(* IEC 61131-3 sources: lacyccom/src/Blocks/Drives, 6 files *)

(* ---- Baseclass.st ---- *)
using System.Timer;
using Siemens.Simatic.DistributedIO;

NAMESPACE Simatic.Ax.LAcycCom

    CLASS ABSTRACT ReadWriteParameter
        VAR
            statrequestBuffer      : Resourcemanager;                                                                                                                  // Connection to the request buffer of the resource manager. All LAcycCom blocks have to use the same request buffer
            statdiagnostics        : LAcycCom_ooptypeDrivediagnostics;                                                                                                 // statdiagnostics structure
            statTimerStart         : BOOL := FALSE;                                                                                                                    // TRUE: Starts IEC-Timer
            statCmdBusy            : BOOL := FALSE;                                                                                                                    // TRUE: Process is NOT yet complete
            statCmdDone            : BOOL := FALSE;                                                                                                                    // TRUE: Data record was transferred
            statCmdError           : BOOL := FALSE;                                                                                                                    // TRUE: An error occurred during processing
            statHwId               : HW_IO := HW_IO#default;                                                                                                           // Intern hardware identifier of the hardware module
            statDoId               : INT;                                                                                                               // Intern identification number of the drive object
            statRefNo              : BYTE := BYTE#16#00;                                                                                                               // Reference number of request
            statFBState            : LAcycCom_ReadWriteStatus := LAcycCom_ReadWriteStatus#FB_IDLE;                                                                     // States in the function block state machine
            statFBSubState         : LAcycCom_ReadWriteStatus := LAcycCom_ReadWriteStatus#FB_BUSY_WRREC;                                                               // States in the function block during processing (busy state)
            statFBSubStateOld      : LAcycCom_ReadWriteStatus := LAcycCom_ReadWriteStatus#FB_BUSY_WRREC;                                                               // Previous state when temporary error occurs
            statStateNumber        : LAcycCom_ReadWriteStatus;                                                                                                         // State of the FB when error occurred
            statDatasetType        : SINT := SINT#0;                                                                                                                   // Dataset type used
            statStatus             : WORD := STATUS_NO_CALL;                                                                                                           // Static value for output status
            statSubfunctionStatus  : WORD := WORD#16#0000;                                                                                                             // Block status OR error information
            statErrorCount         : UINT := UINT#16#0000;                                                                                                             // Error counter of retry request
            statAllocatedIndex     : INT := -1;                                                                                                                        // Allocated element index in the buffer DB
            statCountOfElements    : INT := 0;                                                                                                                         // Number of parameters in the dataset
            statFirstParameterError: INT := -1;                                                                                                                        // Number of parameter at which the error occurred (-1: no parameter with error)
            statDataRecordNo       : DINT;                                                                                                                             // Used data record
            statReqParameter       : LAcycCom_TypestatstatReqParameter;                                                                                                // Request telegram
            statReqParameterInit   : LAcycCom_TypestatparameterAddress :=(attribute := BYTE#16#10, elementNo  := BYTE#16#01, parameterNo := UINT#0, index := UINT#0);

            statRespParameter: LAcycCom_TypestatRespParameter;  // Response telegram
            instWRREC        : WriteRecord;                     // WRREC command
            instRDREC        : ReadRecord;                      // RDREC command
            instIECTimer     : OnDelay;                         // IEC-Timer

            atmpSend : ARRAY[0..237]of BYTE ;
            atmpRec  : ARRAY[0..237]of BYTE ;

         END_VAR

         VAR CONSTANT
            DATA_TYPE_SILENT                    : SINT := SINT#1;        // LAcycCom_typeDriveSilentOperation is in use
            DATA_TYPE_DATASET_REAL              : SINT := SINT#2;        // LAcycCom_typeDriveDatasetReal is in use
            DATA_TYPE_DATASET_DWORD             : SINT := SINT#3;        // LAcycCom_typeDriveDatasetDWord is in use
            NO_PARAMETER_ERROR                  : INT  := INT#-1;        // No parameter error in response telegram
            ALL_ELEMENTS_OCCUPIED               : INT  := INT#-1;        // All buffer elements are occupied
            FORMAT_INTEGER_8                    : SINT := SINT#2;        // Identifier for Integer8 format
            FORMAT_INTEGER_16                   : SINT := SINT#3;        // Identifier for Integer16 format
            FORMAT_INTEGER_32                   : SINT := SINT#4;        // Identifier for Integer32 format
            FORMAT_UNSIGNED_8                   : SINT := SINT#5;        // Identifier for Unsigned8 format
            FORMAT_UNSIGNED_16                  : SINT := SINT#6;        // Identifier for Unsigned16 format
            FORMAT_UNSIGNED_32                  : SINT := SINT#7;        // Identifier for Unsigned32 format
            FORMAT_FLOATING_POINT               : SINT := SINT#8;        // Identifier for Floating Point format
            FORMAT_OCTET_STRING                 : SINT := SINT#10;       // Identifier for OctetString format
            FORMAT_TIME_DIFFERENCE              : SINT := SINT#13;       // Identifier for TimeDifference format
            FORMAT_ZERO                         : SINT := SINT#64;       // Identifier for void telegram
            FORMAT_BYTE                         : SINT := SINT#65;       // Identifier for BYTE format
            FORMAT_WORD                         : SINT := SINT#66;       // Identifier for WORD format
            FORMAT_DOUBLE_WORD                  : SINT := SINT#67;       // Identifier for Double WORD format
            FORMAT_ERROR                        : BYTE := BYTE#16#44;    // Identifier for a format error
            SILENT_OPERATION_PARA_UPPER_LIM     : INT  := 17;            // Maximum count of parameters when using Silent Operation PLC data type
            LENGTH_PARAMETER_TELEGRAM_UPPER_LIM : INT  := 233;           // Maximum length of telegram for parameter information in BYTE
            LENGTH_READ_TELEGRAM_UPPER_LIM      : INT  := 113;           // Maximum length of telegram for parameter information in BYTE
            MAX_ERROR_COUNT                     : UINT := UINT#40;       // Maximum error counter
            TIMER_TEMP_ERROR                    : LTime := T#200MS;       // Waiting time until next system function block call
            TIMER_ALLOCATION                    : LTime := T#10S;         // Timer limit for allocating a request element
            MAX_DRIVE_OBJECT_NO                 : INT  := 254;           // Maximum drive object number limited by SINAMICS p101
            STATUS_EXECUTION_FINISHED           : WORD := WORD#16#0000;  // Execution finished without errors
            STATUS_NO_CALL                      : WORD := WORD#16#7000;  // No call of FB
            STATUS_ALLOCATE                     : WORD := WORD#16#7001;  // FB is currently allocating a request element
            STATUS_GET_RESOURCE                 : WORD := WORD#16#7002;  // FB is waiting until it has “speaking rights”
            STATUS_BUSY                         : WORD := WORD#16#7003;  // FB is currently in processing
            STATUS_RELEASE                      : WORD := WORD#16#7004;  // FB is releasing the allocated element
            WARN_EXECUTE                        : WORD := WORD#16#7100;  // Execute input set during silent operation mode
            ERR_NO_OF_PARAMETERS                : WORD := WORD#16#8001;  // Invalid count of parameters
            ERR_INVALID_PRIORITY_CLASS          : WORD := WORD#16#8002;  // FB is NOT called in OB1
            ERR_REQUEST_REJECTED                : WORD := WORD#16#8004;  // Request rejected
            ERR_RESOURCE_RELEASED               : WORD := WORD#16#8005;  // Request is already released
            ERR_AMBIGUOUS_FB_CALL               : WORD := WORD#16#8006;  // Execute input set during processing (possible inconsistent data at output)
            ERR_INVALID_DATA_TYPE               : WORD := WORD#16#8200;  // Invalid PLC data type at the input "dataset"
            ERR_INVALID_BUF_INDEX               : WORD := WORD#16#8201;  // Buffer index is invalid
            ERR_INVALID_DRIVE_OBJECT_ID         : WORD := WORD#16#8208;  // Drive Object ID is out of range (Drive Object ID < 0 for local access, 1..254 for global access is allowed)
            ERR_COMMAND_TIMEOUT                 : WORD := WORD#16#8600;  // The assigned buffer element is no longer available for the request
            ERR_RDREC_TEMP_COUNTER              : WORD := WORD#16#8601;  // Counter for temporary errors reached the maximum during RDREC command
            ERR_WRREC_TEMP_COUNTER              : WORD := WORD#16#8602;  // Counter for temporary errors reached the maximum during WRREC command
            ERR_WRREC                           : WORD := WORD#16#8603;  // Error occurred during WRREC command
            ERR_RDREC                           : WORD := WORD#16#8604;  // Error occurred during RDREC command
            ERR_REFERENCE_NO                    : WORD := WORD#16#8605;  // Reference number of the request does NOT match the response reference number
            ERR_RESPONSE_ID                     : WORD := WORD#16#8606;  // Invalid response from the drive object
            ERR_PARAMETER_NO                    : WORD := WORD#16#8607;  // The number of parameters received does NOT match the requested number of parameters
            ERR_DRIVE_OBJECT_NO                 : WORD := WORD#16#8608;  // The drive object does NOT match the responded drive object
            ERR_ALLOCATION_TIME                 : WORD := WORD#16#8609;  // The allocation time exceeded the configured value
            ERR_MOVE_BLK_VARIANT                : WORD := WORD#16#8610;  // Error occurred during MOVE_BLK_VARIANT command
            ERR_UNDEFINED_STATE                 : WORD := WORD#16#8611;  // Error due to an undefined state
            ERR_UNDEFINED_SUBSTATE              : WORD := WORD#16#8612;  // Error due to an undefined substate
            ERR_PARAMETER                       : WORD := WORD#16#8619;  // Error in at least one parameter (see: errorValue in dataset)
         END_VAR

        METHOD ABSTRACT BUSY END_METHOD

        METHOD PUBLIC FINAL execute

            //----------------------------------------------------------------------
            // State Machine
            //----------------------------------------------------------------------

            IF NOT (statFBState = LAcycCom_ReadWriteStatus#FB_IDLE OR
                    statFBState = LAcycCom_ReadWriteStatus#FB_DONE OR
                    statFBState = LAcycCom_ReadWriteStatus#FB_ERROR ) THEN  // Functionality running
              CASE statFBState OF
                LAcycCom_ReadWriteStatus#FB_FIRST_CYCLE:  // First cycle state

                    THIS.FIRST_CYCLE();

                    LAcycCom_ReadWriteStatus#FB_ALLOCATE:

                    THIS.Allocate();

                LAcycCom_ReadWriteStatus#FB_GET_RESOURCE:

                    THIS.GET_RESOURCE();

                LAcycCom_ReadWriteStatus#FB_BUSY:

                    THIS.BUSY();

                LAcycCom_ReadWriteStatus#FB_RELEASE:

                    THIS.RELEASE();

                ELSE
                  statStatus := ERR_UNDEFINED_STATE;
                  statStateNumber := statFBState;
                  statFBState := LAcycCom_ReadWriteStatus#FB_ERROR;
              END_CASE;

            END_IF;

            //----------------------------------------------------------------------
            // Error handling and write outputs
            //----------------------------------------------------------------------

            IF (statFBState = LAcycCom_ReadWriteStatus#FB_ERROR) THEN
              // Release the allocated element when error occurs
              IF (statStateNumber <> LAcycCom_ReadWriteStatus#FB_FIRST_CYCLE) AND (statStateNumber <> LAcycCom_ReadWriteStatus#FB_ALLOCATE)
              THEN
                statrequestBuffer.release(statAllocatedIndex);
              END_IF;
              statdiagnostics.stateNumber := statStateNumber;
              statdiagnostics.subfunctionStatus := statSubfunctionStatus;
              statdiagnostics.status := statStatus;

            END_IF;

        END_METHOD

        METHOD FINAL FIRST_CYCLE
            VAR_TEMP
                tempLoopIndex : INT;
                tempVoidDiagnostics : LAcycCom_ooptypeDriveDiagnostics;   // Temporary empty diagnostics structure
                tempVoidHeader : LAcycCom_Typestatheader;   // Temporary empty header structure
             END_VAR

              // Clearing the sending buffer
              statReqParameter.header := tempVoidHeader;
              FOR tempLoopIndex := 0 TO LAcycComConstantsInt#LACYCCOM_READ_PARAMETERS_UPPER_LIM DO
                statReqParameter.parameterAddress[tempLoopIndex] := statReqParameterInit;
              END_FOR;

              // Clearing the receive buffer
              statRespParameter.header := tempVoidHeader;
              FOR tempLoopIndex := 0 TO LENGTH_PARAMETER_TELEGRAM_UPPER_LIM DO
                statRespParameter.data[tempLoopIndex] := BYTE#16#00;
              END_FOR;

              // Initialization after start, depending on the used PLC data type

                IF statDoId < 0 THEN // V1.5
                  statDataRecordNo := 16#B02E; // Base Mode Parameter Access local; doId NOT relevant
                  statDoId := 0; //set DO to zero for use in header
                ELSIF (statDoId <= MAX_DRIVE_OBJECT_NO)
                  AND (statDoId <> 0)
                THEN // V1.5.2
                  statDataRecordNo := 47; // Data record 47; Base Mode Parameter Access global

                ELSE // V1.5.2
                  // Wrong drive object ID at input
                  statStateNumber := statFBState;
                  statStatus := ERR_INVALID_DRIVE_OBJECT_ID;
                  statFBState := LAcycCom_ReadWriteStatus#FB_ERROR;
                END_IF;

                statHwId := statHwId;

              statdiagnostics := tempVoidDiagnostics;
              IF statStatus = WARN_EXECUTE THEN
                statdiagnostics.status := statStatus;
              END_IF;

              statdiagnostics.driveObjectId       := TO_USINT(statDoId);
              statdiagnostics.hardwareId          := statHwId;
              statdiagnostics.firstParameterError := statFirstParameterError;  // V1.3.2
              statdiagnostics.errorValue          := BYTE#16#FF;               // V1.3.2

              // Reference number for next request
              statRefNo := to_byte(to_int(statRefNo) + INT#1);

              IF statFBState = LAcycCom_ReadWriteStatus#FB_ERROR THEN // V1.5.2: Check IF error appeared
                ;

              // Next state is depending on the FB mode
            ELSE
                statStatus := STATUS_ALLOCATE;
                statFBState := LAcycCom_ReadWriteStatus#FB_ALLOCATE;

            END_IF;

        END_METHOD

        METHOD FINAL Allocate
                  // Allocation of a request element
                  statAllocatedIndex := statrequestBuffer.allocate(hardwareId :=statHwId);

                  IF statAllocatedIndex >= 0 THEN

                    statTimerStart := FALSE;
                    statStatus := STATUS_GET_RESOURCE;
                    statFBState := LAcycCom_ReadWriteStatus#FB_GET_RESOURCE;

                  ELSIF (instIECTimer.output = TRUE) THEN
                    statStateNumber := statFBState;
                    statStatus := ERR_ALLOCATION_TIME;
                    statFBState := LAcycCom_ReadWriteStatus#FB_ERROR;

                  ELSE
                    ; // Waiting until lockbit is reset and a request element is available
                  END_IF; // (buffer.lockBuffer = FALSE) AND (buffer.actualWriteIndex >= 0)

                  instIECTimer(signal := statTimerStart,
                                duration := TIMER_ALLOCATION);

                  statTimerStart := TRUE;
                  IF (instIECTimer.output = TRUE) THEN
                    statTimerStart := FALSE;
                  END_IF;
        END_METHOD

        METHOD FINAL GET_RESOURCE
            CASE statrequestBuffer.GetRessource(statAllocatedIndex) of
                // Check buffer index for correctness
                LAcycCom_ResourceManagerRetval#ERR_INVALID_BUF_INDEX:
                  statStateNumber := statFBState;
                  statStatus := ERR_INVALID_BUF_INDEX;
                  statFBState := LAcycCom_ReadWriteStatus#FB_ERROR;

                LAcycCom_ResourceManagerRetval#ERR_REQUEST_REJECTED:
                    // Request was rejected by buffer manager
                    statStateNumber := statFBState;
                    statStatus := ERR_REQUEST_REJECTED;
                    statFBState := LAcycCom_ReadWriteStatus#FB_ERROR;

                LAcycCom_ResourceManagerRetval#ERR_RESOURCE_RELEASED:
                    // Request already released
                    statStateNumber := statFBState;
                    statStatus := ERR_RESOURCE_RELEASED;
                    statFBState := LAcycCom_ReadWriteStatus#FB_ERROR;

                LAcycCom_ResourceManagerRetval#STATUS_BUSY:
                    // Element is enabled
                    statStatus := STATUS_BUSY;
                    statFBState := LAcycCom_ReadWriteStatus#FB_BUSY;
                    statFBSubState := LAcycCom_ReadWriteStatus#FB_GET_SUBSTATE;

                LAcycCom_ResourceManagerRetval#STATUS_GET_RESOURCE:
                    // Element NOT enabled yet
                    //
                    statStatus := STATUS_GET_RESOURCE;
                ELSE
                  ;
                END_CASE;
        end_Method

        METHOD FINAL RELEASE
                  CASE statrequestBuffer.release(statAllocatedIndex) of
                    LAcycCom_ResourceManagerRetval#ERR_INVALID_BUF_INDEX:
                      statStatus := ERR_INVALID_BUF_INDEX;
                      statStateNumber := statFBState;
                      statFBState := LAcycCom_ReadWriteStatus#FB_ERROR;

                    LAcycCom_ResourceManagerRetval#STATUS_EXECUTION_FINISHED:
                      statStatus := STATUS_EXECUTION_FINISHED;
                      statFBState := LAcycCom_ReadWriteStatus#FB_DONE;
                  ELSE
                    ;
                  END_CASE;
        end_Method

        Method PUBLIC FINAL errorDiagnostics   : LAcycCom_ooptypeDrivediagnostics;
            errorDiagnostics := statdiagnostics;
        End_Method

        Method PUBLIC FINAL Status   : LAcycComstateDef;
            CASE statFBState OF
                LAcycCom_ReadWriteStatus#FB_IDLE:
                    Status := LAcycComstateDef#IDLE;

                LAcycCom_ReadWriteStatus#FB_FIRST_CYCLE,
                LAcycCom_ReadWriteStatus#FB_ALLOCATE,
                LAcycCom_ReadWriteStatus#FB_GET_RESOURCE,
                LAcycCom_ReadWriteStatus#FB_BUSY,
                LAcycCom_ReadWriteStatus#FB_RELEASE:
                    Status := LAcycComstateDef#BUSY;

                LAcycCom_ReadWriteStatus#FB_DONE:
                    Status := LAcycComstateDef#DONE;

                LAcycCom_ReadWriteStatus#FB_ERROR:
                    Status := LAcycComstateDef#Error;

                ELSE
                ;
            END_CASE;
        End_Method

        METHOD PUBLIC FINAL Config : BOOL
          VAR_INPUT
              requestBuffer : Resourcemanager;   // Connection to the request buffer of the resource manager. All LAcycCom blocks have to use the same request buffer
           END_VAR

           IF requestBuffer <> NULL THEN
            statrequestBuffer := requestBuffer;
            Config := TRUE;
           ELSE
            ;
           END_IF;

      END_METHOD
    END_CLASS

END_NAMESPACE

(* ---- classReadDriveParams.st ---- *)
using System.Timer;
using siemens.Simatic.DistributedIO;

NAMESPACE Simatic.Ax.LAcycCom
    CLASS LAcycCom_classReadDriveParams EXTENDS ReadWriteParameter
        VAR PRIVATE
            statparameterCount: INT := -1;
            dataset           : Array[0..LAcycComConstantsInt#LACYCCOM_READ_PARAMETERS_UPPER_LIM] of LAcycCom_typeDriveDataset;          // Dataset with all parameters to be read
            statParameter     : Array[0..LAcycComConstantsInt#LACYCCOM_READ_PARAMETERS_UPPER_LIM] of LAcycCom_TypestatstatParameter;     // Parameter dataset
            parameterAddress  : Array[0..LAcycComConstantsInt#LACYCCOM_READ_PARAMETERS_UPPER_LIM] of LAcycCom_TypestatparameterAddress;  // Parameter data in telegram
          END_VAR

        METHOD OVERRIDE BUSY
            VAR_TEMP
                tempCmdValid         : BOOL;                       // TRUE: New data record was received and is valid
                tempStatusWord       : WORD;                       // Temporary status
                tempWord             : WORD;                       // Temporary WORD variable
                tempPointer          : INT;                        // Temporary pointer variable
                tempLoopIndex        : INT;                        // Temporary loop index variable
                tempBlkVariant       : INT;                        // Temporary result of MOVE_BLK_VARIANT
                tempCmdStatus        : DWORD;                      // Temporary status of WRREC and RDREC command
                tempDWord            : DWORD;                      // Temporary DWORD variable
                tempActualElementReal: LAcycCom_typeDriveDataset;  // Temporary element of the dataset (REAL values)
             END_VAR

            IF (statrequestBuffer.GetRessource(statAllocatedIndex)=LAcycCom_ResourceManagerRetval#STATUS_BUSY)
                THEN
                  CASE statFBSubState OF
                    LAcycCom_ReadWriteStatus#FB_GET_SUBSTATE:
                      statFBSubState := LAcycCom_ReadWriteStatus#FB_BUSY_WRREC;

                    LAcycCom_ReadWriteStatus#FB_BUSY_WRREC:  // Writing the dataset configuration into the drive object

                      IF (statCmdBusy = FALSE) THEN
                        // Resets WRREC command
                        instWRREC(request := FALSE,
                                  RECORD := THIS.atmpRec);
                        // Creating header data
                        statReqParameter.header.refNo := statRefNo; // Telegram reference number
                        statReqParameter.header.reqId := BYTE#16#01;  // 0x01 = request parameters
                        statReqParameter.header.doId := TO_BYTE(statDoId);  // Drive object identification number
                        statReqParameter.header.parameterNo := TO_BYTE(statCountOfElements);  // Count of parameters

                        // Copying the dataset into a static variable (depending on the used PLC data type)

                          FOR tempLoopIndex := 0 TO statCountOfElements - 1 DO
                            tempActualElementReal := dataset[tempLoopIndex];

                            statParameter[tempLoopIndex].index := tempActualElementReal.index;
                            statParameter[tempLoopIndex].parameterNo := tempActualElementReal.parameterNumber;
                            statReqParameter.parameterAddress[tempLoopIndex].parameterNo := statParameter[tempLoopIndex].parameterNo;  // Parameter number
                            statReqParameter.parameterAddress[tempLoopIndex].index := statParameter[tempLoopIndex].index;  // Subindex of parameter
                         END_FOR;

                      END_IF; // statCmdBusy = FALSE
                      SerializeBig(UINT#0,
                                  statReqParameter,
                                  THIS.atmpSend );
                      // WRREC command
                      instWRREC(REQUEST := TRUE,                                                 // Transfer data record
                                 hardwareID := statHwId,           // ID number of the hardware component
                                 INDEX  := statDataRecordNo,   // Data record number
                                 LENGTH := UINT#0,             // Maximum length of the data record to be transferred in bytes
                                 DONE   => statCmdDone,        // Data record was transferred
                                 BUSY   => statCmdBusy,        // The writing process is NOT yet complete
                                 ERROR  => statCmdError,       // An error occurred during the writing process
                                 STATUS => tempCmdStatus,      // Status[1] = Error => Status[2] Error Decode + Status[3] Error Code
                                 RECORD := THIS.atmpSend);     // Data record

                      // Error occurred
                      IF (statCmdError = TRUE) AND NOT(statFBState = LAcycCom_ReadWriteStatus#FB_ERROR) THEN
                        tempStatusWord.%B0 := tempCmdStatus.%B1;
                        tempStatusWord.%B1 := tempCmdStatus.%B2;

                        //Temporary command status (80A1, 80A7, 80B5, 80C0, 80C1, 80C2, 80C3 oder 80C4) are valid and retry command
                        IF (tempStatusWord = WORD#16#80A1) OR  // Negative acknowledgment when writing to the module
                          (tempStatusWord = WORD#16#80A7) OR   // DP slave OR module is occupied (temporary error)
                          (tempStatusWord = WORD#16#80B5) OR   // DP slave OR module NOT ready
                          (tempStatusWord = WORD#16#80C0) OR   // The data can only be written when the CPU is in STOP mode. Note: this means that writing by the user program is NOT possible. You can only write the data online with PG/PC.
                          (tempStatusWord = WORD#16#80C1) OR   // The data of the previous write job on the module for the same data record have NOT yet been processed by the module.
                          (tempStatusWord = WORD#16#80C2) OR   // The module is currently processing the maximum possible number of jobs for a CPU.
                          (tempStatusWord = WORD#16#80C3) OR   // The required operating resources are currently occupied.
                          (tempStatusWord = WORD#16#80C4) THEN // Internal temporary error. Job could NOT be executed. Repeat the job. IF this error occurs often, check your installation for sources of electrical interference.

                          IF (statErrorCount >= MAX_ERROR_COUNT) THEN
                            statStateNumber := statFBSubState;
                            statSubfunctionStatus := tempStatusWord;
                            statStatus := ERR_WRREC_TEMP_COUNTER;
                            statFBState := LAcycCom_ReadWriteStatus#FB_ERROR;
                          ELSE
                            statErrorCount := statErrorCount + UINT#1;  // Increment internal error counter
                            statFBSubStateOld := LAcycCom_ReadWriteStatus#FB_BUSY_WRREC;
                            statFBSubState := LAcycCom_ReadWriteStatus#FB_BUSY_WAIT;
                          END_IF;
                        ELSE
                          statStateNumber := statFBSubState;
                          statSubfunctionStatus := tempStatusWord;
                          statStatus := ERR_WRREC;
                          statFBState := LAcycCom_ReadWriteStatus#FB_ERROR;
                        END_IF;

                      ELSIF (statCmdDone = TRUE) AND NOT(statFBState = LAcycCom_ReadWriteStatus#FB_ERROR) THEN  // Processing completed without errors
                        statErrorCount := UINT#0;  // V1.5.1 Reset error counter
                        statFBSubState := LAcycCom_ReadWriteStatus#FB_BUSY_RDREC; // WRREC completed and continue with RDREC
                      END_IF; // statCmdError = TRUE

                      LAcycCom_ReadWriteStatus#FB_BUSY_RDREC:  // Reading the values from the drive object
                      // Resets RDREC command
                      IF (statCmdBusy = FALSE) THEN
                        instRDREC(REQUEST := FALSE,
                                   RECORD := THIS.atmpRec);
                      END_IF;

                      instRDREC(REQUEST := TRUE,                                                 // Transfer data record
                                 hardwareID := statHwId,           // ID number of the hardware component
                                 INDEX      := statDataRecordNo,   // Data record number
                                 MAXLENGTH  := UINT#0,             // Maximum length in bytes of the data record information to be read
                                 VALID      => tempCmdValid,       // New data record was received and is valid
                                 BUSY       => statCmdBusy,        // The reading process is NOT yet complete
                                 ERROR      => statCmdError,       // An error occurred during the reading process
                                 STATUS     => tempCmdStatus,      // Status[1] = Error => Status[2] Error Decode + Status[3] Error Code
                                 RECORD     := THIS.atmpRec);      // Destination area for the data record read

                      DeserializeBig(UINT#0,
                                 THIS.atmpRec,
                                 statRespParameter);
                      // Error occurred
                      IF (statCmdError = TRUE) THEN
                        // Get the error information from the status information
                        tempStatusWord.%B0 := tempCmdStatus.%B1;
                        tempStatusWord.%B1 := tempCmdStatus.%B2;

                        //Temporary command status (80A0, 80A7, 80B5, 80C0, 80C1, 80C2, 80C3 oder 80C4) are valid and retry command
                        IF (tempStatusWord = WORD#16#80A0) OR  // Negative acknowledgment when reading the module
                          (tempStatusWord = WORD#16#80A7) OR   // DP slave OR module is occupied (temporary error)
                          (tempStatusWord = WORD#16#80B5) OR   // DP slave OR module NOT ready
                          (tempStatusWord = WORD#16#80C0) OR   // The data can only be written when the CPU is in STOP mode. Note: this means that writing by the user program is NOT possible. You can only write the data online with PG/PC.
                          (tempStatusWord = WORD#16#80C1) OR   // The data of the previous write job on the module for the same data record have NOT yet been processed by the module.
                          (tempStatusWord = WORD#16#80C2) OR   // The module is currently processing the maximum possible number of jobs for a CPU.
                          (tempStatusWord = WORD#16#80C3) OR   // The required operating resources are currently occupied.
                          (tempStatusWord = WORD#16#80C4) THEN // Internal temporary error. Job could NOT be executed. Repeat the job. IF this error occurs often, check your installation for sources of electrical interference.

                          IF (statErrorCount >= MAX_ERROR_COUNT) THEN
                            statStateNumber := statFBSubState;
                            statSubfunctionStatus := tempStatusWord;
                            statStatus := ERR_RDREC_TEMP_COUNTER;
                            statFBState := LAcycCom_ReadWriteStatus#FB_ERROR;
                          ELSE
                            statErrorCount := statErrorCount + UINT#1;  // Increment internal error counter
                            statFBSubStateOld := LAcycCom_ReadWriteStatus#FB_BUSY_RDREC;
                            // V1.3.2. IF error 80A0 THEN should be retry with WRREC command
                            IF (tempStatusWord = WORD#16#80A0) THEN
                              statFBSubStateOld := LAcycCom_ReadWriteStatus#FB_BUSY_WRREC;
                            END_IF;
                            statFBSubState := LAcycCom_ReadWriteStatus#FB_BUSY_WAIT;
                          END_IF; // statErrorCount >= MAX_ERROR_COUNT
                        ELSE
                          statStateNumber := statFBSubState;
                          statSubfunctionStatus := tempStatusWord;
                          statStatus := ERR_RDREC;
                          statFBState := LAcycCom_ReadWriteStatus#FB_ERROR;
                        END_IF;

                        // Error : Reference number of the request does NOT match with the response reference number
                      ELSIF (statCmdBusy = FALSE) AND
                        (statRefNo <> statRespParameter.header.refNo) AND
                        (tempCmdValid = TRUE) THEN

                        statStateNumber := statFBSubState;
                        statStatus := ERR_REFERENCE_NO;
                        statFBState := LAcycCom_ReadWriteStatus#FB_ERROR;

                        // Error : Invalid response from the drive object (reqId: 16#01 - reading parameter successful; 16#81: reading parameter finished with error)
                      ELSIF NOT (statRespParameter.header.reqId = BYTE#16#81 OR statRespParameter.header.reqId = BYTE#16#01) AND
                        (statCmdBusy = FALSE) AND
                        (tempCmdValid = TRUE) THEN
                        statStateNumber := statFBSubState;
                        statStatus := ERR_RESPONSE_ID;
                        statFBState := LAcycCom_ReadWriteStatus#FB_ERROR;

                        // Error : The received number of parameters does NOT match with the requested number of parameters
                      ELSIF (statCmdBusy = FALSE) AND
                        (statCountOfElements <> TO_INT(statRespParameter.header.parameterNo)) AND
                        (tempCmdValid = TRUE) THEN

                        statStateNumber := statFBSubState;
                        statStatus := ERR_PARAMETER_NO;
                        statFBState := LAcycCom_ReadWriteStatus#FB_ERROR;

                        // Error : The drive object does NOT match with the responsed DO
                      ELSIF (statCmdBusy = FALSE) AND
                        (TO_BYTE(statDoId) <> statRespParameter.header.doId) AND
                        (tempCmdValid = TRUE) THEN

                        statStateNumber := statFBSubState;
                        statStatus := ERR_DRIVE_OBJECT_NO;
                        statFBState := LAcycCom_ReadWriteStatus#FB_ERROR;

                        // No error occurred during reading parameters
                      ELSIF (tempCmdValid = TRUE) THEN
                        // Analyse of the response buffer
                        tempPointer := 0;
                        FOR tempLoopIndex := 0 TO statCountOfElements - 1 DO
                          statParameter[tempLoopIndex].format := statRespParameter.data[tempPointer];  // Format of the parameter

                          // Format = Error
                          IF (((TO_SINT(statRespParameter.data[tempPointer]) > FORMAT_DOUBLE_WORD) OR
                            ((TO_SINT(statRespParameter.data[tempPointer]) > FORMAT_FLOATING_POINT) AND (TO_SINT(statRespParameter.data[tempPointer]) < FORMAT_OCTET_STRING)) OR
                            ((TO_SINT(statRespParameter.data[tempPointer]) > FORMAT_OCTET_STRING) AND (TO_SINT(statRespParameter.data[tempPointer]) < FORMAT_TIME_DIFFERENCE)) OR
                            ((TO_SINT(statRespParameter.data[tempPointer]) > FORMAT_TIME_DIFFERENCE) AND (TO_SINT(statRespParameter.data[tempPointer]) < FORMAT_BYTE)) OR
                            (TO_SINT(statRespParameter.data[tempPointer]) < FORMAT_INTEGER_8))) AND (TO_SINT(statRespParameter.data[tempPointer]) <> FORMAT_ZERO)
                          THEN

                            // Format = Error, summarize the first and second error BYTE in a WORD error variable for each parameter
                            statParameter[tempLoopIndex].errorValue := statRespParameter.data[tempPointer + 3];
                            IF (statFirstParameterError = NO_PARAMETER_ERROR) THEN
                              statdiagnostics.firstParameterError := tempLoopIndex;
                              statdiagnostics.errorValue := statParameter[tempLoopIndex].errorValue; // V1.3.2
                              statFirstParameterError := tempLoopIndex;
                              statStateNumber := statFBSubState;
                              statStatus := ERR_PARAMETER;
                              statFBState := LAcycCom_ReadWriteStatus#FB_ERROR;
                            END_IF;
                            // Points to the next parameter address
                            tempPointer := tempPointer + 6;

                          ELSE

                            CASE TO_SINT(statRespParameter.data[tempPointer]) OF
                              FORMAT_INTEGER_8:

                                  statParameter[tempLoopIndex].realValue := TO_REAL(TO_SINT(statRespParameter.data[tempPointer + 2]));
                                  statParameter[tempLoopIndex].dwordValue := statRespParameter.data[tempPointer + 2];

                                statParameter[tempLoopIndex].errorValue := BYTE#16#FF; // Sets the error status and diagnostics
                                tempPointer := tempPointer + 4; // Points to the next parameter address

                              FORMAT_INTEGER_16:
                                tempWord.%B0 := statRespParameter.data[tempPointer + 3];
                                tempWord.%B1 := statRespParameter.data[tempPointer + 2];

                                statParameter[tempLoopIndex].realValue := TO_REAL(TO_INT(tempWord));
                                statParameter[tempLoopIndex].dwordValue := tempWord;
                                statParameter[tempLoopIndex].errorValue := BYTE#16#FF; // Sets the error status and diagnostics
                                tempPointer := tempPointer + 4; // Points to the next parameter address

                              FORMAT_INTEGER_32:
                                tempDWord.%B0 := statRespParameter.data[tempPointer + 5];
                                tempDWord.%B1 := statRespParameter.data[tempPointer + 4];
                                tempDWord.%B2 := statRespParameter.data[tempPointer + 3];
                                tempDWord.%B3 := statRespParameter.data[tempPointer + 2];

                                statParameter[tempLoopIndex].realValue := TO_REAL(TO_DINT(tempDWord));
                                statParameter[tempLoopIndex].dwordValue := tempDWord;

                                statParameter[tempLoopIndex].errorValue := BYTE#16#FF; // Sets the error status and diagnostics
                                tempPointer := tempPointer + 6; // Points to the next parameter address

                              FORMAT_UNSIGNED_8, FORMAT_OCTET_STRING: // V1.5 change OCTET_STRING

                                statParameter[tempLoopIndex].realValue := TO_REAL(TO_USINT(statRespParameter.data[tempPointer + 2]));
                                statParameter[tempLoopIndex].dwordValue := statRespParameter.data[tempPointer + 2];

                                statParameter[tempLoopIndex].errorValue := BYTE#16#FF; // Sets the error status and diagnostics
                                tempPointer := tempPointer + 4; // Points to the next parameter address
                              FORMAT_UNSIGNED_16:
                                tempWord.%B0 := statRespParameter.data[tempPointer + 3];
                                tempWord.%B1 := statRespParameter.data[tempPointer + 2];

                                statParameter[tempLoopIndex].realValue := TO_REAL(TO_UINT(tempWord));
                                statParameter[tempLoopIndex].dwordValue := tempWord;

                                statParameter[tempLoopIndex].errorValue := BYTE#16#FF; // Sets the error status and diagnostics
                                tempPointer := tempPointer + 4; // Points to the next parameter address

                              FORMAT_UNSIGNED_32, FORMAT_TIME_DIFFERENCE:
                                tempDWord.%B0 := statRespParameter.data[tempPointer + 5];
                                tempDWord.%B1 := statRespParameter.data[tempPointer + 4];
                                tempDWord.%B2 := statRespParameter.data[tempPointer + 3];
                                tempDWord.%B3 := statRespParameter.data[tempPointer + 2];

                                statParameter[tempLoopIndex].realValue := TO_REAL(TO_UDINT(tempDWord));
                                statParameter[tempLoopIndex].dwordValue := tempDWord;

                                statParameter[tempLoopIndex].errorValue := BYTE#16#FF; // Sets the error status and diagnostics
                                tempPointer := tempPointer + 6; // Points to the next parameter address

                              FORMAT_FLOATING_POINT, FORMAT_DOUBLE_WORD:
                                tempDWord.%B0 := statRespParameter.data[tempPointer + 5];
                                tempDWord.%B1 := statRespParameter.data[tempPointer + 4];
                                tempDWord.%B2 := statRespParameter.data[tempPointer + 3];
                                tempDWord.%B3 := statRespParameter.data[tempPointer + 2];

                                statParameter[tempLoopIndex].realValue := TO_REAL(tempDWord);
                                statParameter[tempLoopIndex].dwordValue := tempDWord;

                                statParameter[tempLoopIndex].errorValue := BYTE#16#FF; // Sets the error status and diagnostics
                                tempPointer := tempPointer + 6; // Points to the next parameter address

                              FORMAT_BYTE:
                                statParameter[tempLoopIndex].realValue := TO_REAL(TO_DWORD(statRespParameter.data[tempPointer + 2]));
                                statParameter[tempLoopIndex].dwordValue := statRespParameter.data[tempPointer + 2];

                                statParameter[tempLoopIndex].errorValue := BYTE#16#FF; // Sets the error status and diagnostics
                                tempPointer := tempPointer + 4; // Points to the next parameter address

                              FORMAT_WORD:
                                tempWord.%B0 := statRespParameter.data[tempPointer + 3];
                                tempWord.%B1 := statRespParameter.data[tempPointer + 2];

                                statParameter[tempLoopIndex].realValue := TO_REAL(TO_DWORD(tempWord));
                                statParameter[tempLoopIndex].dwordValue := tempWord;

                                statParameter[tempLoopIndex].errorValue := BYTE#16#FF; // Sets the error status and diagnostics
                                tempPointer := tempPointer + 4; // Points to the next parameter address

                              ELSE
                                ;
                            END_CASE;

                          END_IF; // Format = Error
                        END_FOR; // Analyse of the response buffer

                        // Copying parameter data into the dataset (depending on the used PLC data type)

                          FOR tempLoopIndex := 0 TO statCountOfElements - 1 BY 1 DO
                            tempActualElementReal.index := statParameter[tempLoopIndex].index;
                            tempActualElementReal.parameterNumber := statParameter[tempLoopIndex].parameterNo;
                            tempActualElementReal.Rvalue := statParameter[tempLoopIndex].realValue;
                            tempActualElementReal.DWvalue := statParameter[tempLoopIndex].dwordValue;
                            tempActualElementReal.errorValue := statParameter[tempLoopIndex].errorValue;
                           // tempBlkVariant := MOVE_BLK_VARIANT(SRC := tempActualElementReal, COUNT := 1, SRC_INDEX := 0, DEST_INDEX := tempLoopIndex, DEST => dataset);
                            dataset[tempLoopIndex] := tempActualElementReal;
                            // Error occurred during MOVE_BLK_VARIANT command
                            IF (tempBlkVariant <> 0) THEN
                              statStateNumber := statFBSubState;
                              statSubfunctionStatus := TO_WORD(tempBlkVariant);
                              statStatus := ERR_MOVE_BLK_VARIANT;
                              statFBState := LAcycCom_ReadWriteStatus#FB_ERROR;
                              statdiagnostics.firstParameterError := tempLoopIndex;
                            END_IF;
                          END_FOR;

                        // Next state is depending on the FB mode
                        IF NOT(statFBState = LAcycCom_ReadWriteStatus#FB_ERROR) THEN
                          statStatus := STATUS_RELEASE;
                          statFBState := LAcycCom_ReadWriteStatus#FB_RELEASE;

                        END_IF; // statMode = MODE_WITH_BUFFER_MANAGER
                      END_IF; // statCmdError = TRUE

                      LAcycCom_ReadWriteStatus#FB_BUSY_WAIT:
                      // Timer for temporary errors
                      instIECTimer(signal := statTimerStart,
                                    duration := TIMER_TEMP_ERROR);

                      statTimerStart := TRUE;
                      IF (instIECTimer.output = TRUE) THEN
                        statTimerStart := FALSE;
                        statFBSubState := statFBSubStateOld;
                      END_IF;

                    ELSE
                      statStatus := ERR_UNDEFINED_SUBSTATE;
                      statStateNumber := statFBState;
                      statFBState := LAcycCom_ReadWriteStatus#FB_ERROR;
                  END_CASE;

                ELSE
                  statStatus := ERR_COMMAND_TIMEOUT;
                  statStateNumber := statFBState;
                  statFBState := LAcycCom_ReadWriteStatus#FB_ERROR;
                END_IF; // ((buffer.element[statAllocatedIndex].enable = TRUE) AND (statMode = MODE_WITH_BUFFER_MANAGER)) OR statMode = MODE_WITHOUT_BUFFER_MANAGER

        END_METHOD

                //data type of driveobjectid has been changed from uint to int. This extra start method keeps compability to old versions of LAcycCom
                METHOD PUBLIC Start : BOOL
                  VAR_INPUT
                    driveObjectId : UINT;
                    hardwareId    : HW_IO;
                    parameterCount: INT := -1;
                  END_VAR
                  Start := THIS.Start(driveObjectId := TO_INT(driveObjectId), hardwareId := hardwareId, parameterCount := parameterCount);
                END_METHOD
                //data type of driveobjectid has been changed from uint to int. This extra start method can be used, if direct hw id is used and drive object is not used (equivalent to driveobjectid = -1)
                METHOD PUBLIC Start : BOOL
                  VAR_INPUT
                    hardwareId    : HW_IO;
                    parameterCount: INT := -1;
                END_VAR
                Start := THIS.Start(driveObjectId := -1, hardwareId := hardwareId, parameterCount := parameterCount);
              END_METHOD

        METHOD PUBLIC Start : BOOL
            VAR_INPUT
              driveObjectId  : INT := -1;   // Optional: Identification number of the drive object (value =-1: driveObjectId is NOT used, i.e. the corresponding drive object is only addressed via the hardwareId)
              hardwareId : HW_IO;   // Hardware identifier of the hardware module
              parameterCount : INT := -1;   // Count of parameters to read (-1: read all parameter in dataset)
            END_VAR

             statparameterCount := parameterCount;
             statDoId := driveObjectId;
             statHwId := hardwareId;

             // starts functionality
             IF NOT ((statFBState = LAcycCom_ReadWriteStatus#FB_IDLE OR
                 statFBState = LAcycCom_ReadWriteStatus#FB_DONE OR
                 statFBState = LAcycCom_ReadWriteStatus#FB_ERROR) AND
                 statrequestBuffer <> NULL) THEN
                   Start := FALSE;
             ELSE
               // Initialisation
               Start := TRUE;
               statAllocatedIndex := -1;
               statSubfunctionStatus :=  WORD#16#0000;
               statDataRecordNo := DINT#0;
               statStateNumber := LAcycCom_ReadWriteStatus#FB_IDLE;
               statDatasetType := SINT#0;
               statFirstParameterError := -1;
               statErrorCount := UINT#0;
               statFBSubState := LAcycCom_ReadWriteStatus#FB_BUSY_WRREC;
               statFBState := LAcycCom_ReadWriteStatus#FB_FIRST_CYCLE;

               instIECTimer(signal := FALSE,
                             duration := TIMER_ALLOCATION);
             END_IF;
        END_METHOD

        Method PUBLIC DeleteList
            Var
                z : INT;
            END_VAR

            For z := 0 to LAcycComConstantsInt#LACYCCOM_READ_PARAMETERS_UPPER_LIM do
                dataset[z].DWvalue         := DWORD#0;
                dataset[z].errorValue      := BYTE#0;
                dataset[z].index           := UINT#0;
                dataset[z].parameterNumber := UINT#0;
                dataset[z].Rvalue          := REAL#0.0;
            end_FOR;
            statCountOfElements := 0;
        End_Method

        Method PUBLIC AddatasetItem : INT //Rückgabewert = anzahl der Listeneinträge
            VAR_INPUT
                datasetItem : LAcycCom_typeDriveDataset;
                element_no  : INT := INT#-1; //-1 element an die liste anhängen. >=0 element überschreiben
            END_VAR
            VAR_TEMP
                tempLoopIndex : INT;
            END_VAR
            IF element_no = -1 and statCountOfElements < LAcycComConstantsInt#LACYCCOM_READ_PARAMETERS_UPPER_LIM THEN
                    dataset[statCountOfElements] :=datasetItem;
                statCountOfElements := statCountOfElements + 1;
                AddatasetItem := statCountOfElements;

            elsif element_no > -1 and
                element_no < LAcycComConstantsInt#LACYCCOM_READ_PARAMETERS_UPPER_LIM and
                element_no <= statCountOfElements THEN
                    dataset[element_no] :=datasetItem;
                    IF element_no = statCountOfElements THEN
                        statCountOfElements := statCountOfElements + 1;
                    END_IF;
                    AddatasetItem := statCountOfElements;
            ELSE
                AddatasetItem := -1;
            END_IF;

        End_Method

        Method PUBLIC ReaddatasetItem : LAcycCom_typeDriveDataset
            VAR_INPUT
                element_no  : INT := INT#0;
            END_VAR
            VAR_TEMP
                tempLoopIndex : INT;
            END_VAR

            IF element_no >= 0 and element_no <= LAcycComConstantsInt#LACYCCOM_READ_PARAMETERS_UPPER_LIM THEN
                ReaddatasetItem := dataset[element_no];
            END_IF;

        End_Method

        Method PUBLIC ReaddatasetValue : REAL
          VAR_INPUT
              element_no  : INT := INT#0;
          END_VAR
          VAR_TEMP
              tempLoopIndex : INT;
          END_VAR

          IF element_no >= 0 and element_no <= LAcycComConstantsInt#LACYCCOM_READ_PARAMETERS_UPPER_LIM THEN
            ReaddatasetValue := dataset[element_no].Rvalue;
          END_IF;

        End_Method

        Method PUBLIC ReaddatasetDWValue : DWORD
          VAR_INPUT
              element_no  : INT := INT#0;
          END_VAR
          VAR_TEMP
              tempLoopIndex : INT;
          END_VAR

          IF element_no >= 0 and element_no <= LAcycComConstantsInt#LACYCCOM_READ_PARAMETERS_UPPER_LIM THEN
            ReaddatasetDWValue := dataset[element_no].DWvalue;
          END_IF;

        End_Method

    END_CLASS
END_NAMESPACE

(* ---- classReadDriveSingleParams.st ---- *)
using System.Timer;
using siemens.Simatic.DistributedIO;

NAMESPACE Simatic.Ax.LAcycCom
    CLASS LAcycCom_classReadDriveSingleParams EXTENDS ReadWriteParameter
        VAR PRIVATE
            statparameterNumber: UINT;                                                                      // Number of the parameter
            statindex          : UINT;                                                                      // Parameter index
            statParameter      : Array[0..READ_PARAMETERS_UPPER_LIM] of LAcycCom_TypestatstatParameter;     // Parameter dataset
            parameterAddress   : Array[0..READ_PARAMETERS_UPPER_LIM] of LAcycCom_TypestatparameterAddress;  // Parameter data in telegram
        END_VAR

        VAR CONSTANT
          READ_PARAMETERS_UPPER_LIM : INT := 0;
        END_VAR

        METHOD OVERRIDE BUSY
            VAR_TEMP
                tempCmdValid         : BOOL;                       // TRUE: New data record was received and is valid
                tempStatusWord       : WORD;                       // Temporary status
                tempWord             : WORD;                       // Temporary WORD variable
                tempPointer          : INT;                        // Temporary pointer variable
                tempLoopIndex        : INT;                        // Temporary loop index variable
                tempBlkVariant       : INT;                        // Temporary result of MOVE_BLK_VARIANT
                tempCmdStatus        : DWORD;                      // Temporary status of WRREC and RDREC command
                tempDWord            : DWORD;                      // Temporary DWORD variable
                tempVoidHeader       : LAcycCom_Typestatheader;    // Temporary empty header structure
                tempActualElementReal: LAcycCom_typeDriveDataset;  // Temporary element of the dataset (REAL values)
             END_VAR
             IF (statrequestBuffer.GetRessource(statAllocatedIndex)=LAcycCom_ResourceManagerRetval#STATUS_BUSY) THEN

               CASE statFBSubState OF
                LAcycCom_ReadWriteStatus#FB_GET_SUBSTATE:
                    statFBSubState := LAcycCom_ReadWriteStatus#FB_BUSY_WRREC;

                LAcycCom_ReadWriteStatus#FB_BUSY_WRREC:  // Writing the dataset configuration into the drive object

                   IF  (statCmdBusy = FALSE) THEN
                     // Resets WRREC command
                     instWRREC(request := FALSE,
                               RECORD := THIS.atmpSend);

                     // Creating header data
                     statReqParameter.header.refNo := statRefNo; // Telegram reference number
                     statReqParameter.header.reqId := BYTE#16#01;  // 0x01 = request parameters
                     statReqParameter.header.doId := TO_BYTE(statDoId);  // Drive object identification number
                     statReqParameter.header.parameterNo := BYTE#16#01;  // Count of parameters

                     // Copying the dataset into a static variable
                     statParameter[tempLoopIndex].index := statindex;
                     statParameter[tempLoopIndex].parameterNo := statParameterNumber;
                     statReqParameter.parameterAddress[tempLoopIndex].parameterNo := statParameter[tempLoopIndex].parameterNo;  // Parameter number
                     statReqParameter.parameterAddress[tempLoopIndex].index := statParameter[tempLoopIndex].index;  // Subindex of parameter

                   END_IF; // statCmdBusy = FALSE

                   // WRREC command
                 SerializeBig(UINT#0,
                             statReqParameter,
                             THIS.atmpSend );

                   instWRREC(REQUEST := TRUE,                                                 // Transfer data record
                              hardwareID := statHwId,           // ID number of the hardware component
                              INDEX      := statDataRecordNo,   // Data record number
                              LENGTH     := UINT#0,             // Maximum length of the data record to be transferred in bytes
                              DONE       => statCmdDone,        // Data record was transferred
                              BUSY       => statCmdBusy,        // The writing process is NOT yet complete
                              ERROR      => statCmdError,       // An error occurred during the writing process
                              STATUS     => tempCmdStatus,      // Status[1] = Error => Status[2] Error Decode + Status[3] Error Code
                              RECORD     := THIS.atmpSend);     // Data record

                   // Error occurred
                   IF  (statCmdError = TRUE) AND   NOT(statFBState = LAcycCom_ReadWriteStatus#FB_ERROR) THEN
                     tempStatusWord.%B0 := tempCmdStatus.%B1;
                     tempStatusWord.%B1 := tempCmdStatus.%B2;

                     // Temporary command status (80A1, 80A7, 80B5, 80C0, 80C1, 80C2, 80C3 oder 80C4) are valid and retry command
                     IF  (tempStatusWord = WORD#16#80A1) OR  // Negative acknowledgment when writing to the module
                        (tempStatusWord = WORD#16#80A7) OR   // DP slave OR module is occupied (temporary error)
                        (tempStatusWord = WORD#16#80B5) OR   // DP slave OR module NOT ready
                        (tempStatusWord = WORD#16#80C0) OR   // The data can only be written when the CPU is in STOP mode. Note: this means that writing by the user program is NOT possible. You can only write the data online with PG/PC.
                        (tempStatusWord = WORD#16#80C1) OR   // The data of the previous write job on the module for the same data record have NOT yet been processed by the module.
                        (tempStatusWord = WORD#16#80C2) OR   // The module is currently processing the maximum possible number of jobs for a CPU.
                        (tempStatusWord = WORD#16#80C3) OR   // The required operating resources are currently occupied.
                        (tempStatusWord = WORD#16#80C4) THEN // Internal temporary error. Job could NOT be executed. Repeat the job. IF this error occurs often, check your installation for sources of electrical interference.

                       IF  (statErrorCount >= MAX_ERROR_COUNT) THEN

                         statStateNumber := statFBSubState;
                         statSubfunctionStatus := tempStatusWord;
                         statStatus := ERR_WRREC_TEMP_COUNTER;
                         statFBState :=  LAcycCom_ReadWriteStatus#FB_ERROR;
                       ELSE
                         statErrorCount := statErrorCount + UINT#1;  // Increment internal error counter
                         statFBSubStateOld := LAcycCom_ReadWriteStatus#FB_BUSY_WRREC;
                         statFBSubState := LAcycCom_ReadWriteStatus#FB_BUSY_WAIT;
                       END_IF;
                     ELSE

                       statStateNumber := statFBSubState;
                       statSubfunctionStatus := tempStatusWord;
                       statStatus := ERR_WRREC;
                       statFBState :=  LAcycCom_ReadWriteStatus#FB_ERROR;
                     END_IF;

                   ELSIF  (statCmdDone = TRUE) AND   NOT(statFBState = LAcycCom_ReadWriteStatus#FB_ERROR) THEN  // Processing completed without errors
                     statFBSubState := LAcycCom_ReadWriteStatus#FB_BUSY_RDREC; // WRREC completed and continue with RDREC
                     statErrorCount := UINT#0;  // V1.5.1 Reset error counter
                   END_IF; // statCmdError = TRUE

                   LAcycCom_ReadWriteStatus#FB_BUSY_RDREC:  // Reading the values from the drive object
                   // Resets RDREC command
                   IF  (statCmdBusy = FALSE) THEN
                     instRDREC(request := FALSE,
                                RECORD := THIS.atmpRec);
                   END_IF;

                   instRDREC(REQUEST := TRUE,                                                 // Transfer data record
                              hardwareID := statHwId,                                                 // ID number of the hardware component
                              INDEX := statDataRecordNo,                                      // Data record number
                              MAXLENGTH := UINT#0,                                            // Maximum length in bytes of the data record information to be read
                              VALID => tempCmdValid,                                          // New data record was received and is valid
                              BUSY => statCmdBusy,                                            // The reading process is NOT yet complete
                              ERROR => statCmdError,                                          // An error occurred during the reading process
                              STATUS => tempCmdStatus,                                        // Status[1] = Error => Status[2] Error Decode + Status[3] Error Code
                              RECORD := THIS.atmpRec);                                             // Destination area for the data record read

                             DeserializeBig(UINT#0,
                              THIS.atmpRec,
                              statRespParameter);

                               // Destination aapaarea for the data record read

                   // Error occurred
                   IF  (statCmdError = TRUE) THEN
                     // Get the error information from the status information
                     tempStatusWord.%B0 := tempCmdStatus.%B1;
                     tempStatusWord.%B1 := tempCmdStatus.%B2;

                     // Temporary command status (80A0, 80A7, 80B5, 80C0, 80C1, 80C2, 80C3 oder 80C4) are valid and retry command
                     IF  (tempStatusWord = WORD#16#80A0) OR  // Negative acknowledgment when reading the module
                        (tempStatusWord = WORD#16#80A7) OR   // DP slave OR module is occupied (temporary error)
                        (tempStatusWord = WORD#16#80B5) OR   // DP slave OR module NOT ready
                        (tempStatusWord = WORD#16#80C0) OR   // The data can only be written when the CPU is in STOP mode. Note: this means that writing by the user program is NOT possible. You can only write the data online with PG/PC.
                        (tempStatusWord = WORD#16#80C1) OR   // The data of the previous write job on the module for the same data record have NOT yet been processed by the module.
                        (tempStatusWord = WORD#16#80C2) OR   // The module is currently processing the maximum possible number of jobs for a CPU.
                        (tempStatusWord = WORD#16#80C3) OR   // The required operating resources are currently occupied.
                        (tempStatusWord = WORD#16#80C4) THEN // Internal temporary error. Job could NOT be executed. Repeat the job. IF this error occurs often, check your installation for sources of electrical interference.

                       IF  (statErrorCount >= MAX_ERROR_COUNT) THEN

                         statStateNumber := statFBSubState;
                         statSubfunctionStatus := tempStatusWord;
                         statStatus := ERR_RDREC_TEMP_COUNTER;
                         statFBState :=  LAcycCom_ReadWriteStatus#FB_ERROR;
                       ELSE
                         statErrorCount := statErrorCount + UINT#1;  // Increment internal error counter
                         statFBSubStateOld := LAcycCom_ReadWriteStatus#FB_BUSY_RDREC;
                         // V1.3.2. IF error 80A0 THEN should be retry with WRREC command
                         IF  (tempStatusWord = WORD#16#80A0) THEN
                           statFBSubStateOld := LAcycCom_ReadWriteStatus#FB_BUSY_WRREC;
                         END_IF;
                         statFBSubState := LAcycCom_ReadWriteStatus#FB_BUSY_WAIT;
                       END_IF; // statErrorCount >= MAX_ERROR_COUNT
                     ELSE

                       statStateNumber := statFBSubState;
                       statSubfunctionStatus := tempStatusWord;
                       statStatus := ERR_RDREC;
                       statFBState :=  LAcycCom_ReadWriteStatus#FB_ERROR;
                     END_IF;

                     // Error : Reference number of the request does NOT match with the response reference number
                   ELSIF  (statCmdBusy = FALSE) AND
                      (statRefNo <> statRespParameter.header.refNo) AND
                      (tempCmdValid = TRUE) THEN

                     statStateNumber := statFBSubState;
                     statStatus := ERR_REFERENCE_NO;
                     statFBState :=  LAcycCom_ReadWriteStatus#FB_ERROR;

                     // Error : Invalid response from the drive object (reqId: 16#01 - reading parameter successful; 16#81: reading parameter finished with error)
                   ELSIF NOT  (statRespParameter.header.reqId = BYTE#16#81 OR statRespParameter.header.reqId = BYTE#16#01) AND
                      (statCmdBusy = FALSE) AND
                      (tempCmdValid = TRUE) THEN

                     statStateNumber := statFBSubState;
                     statStatus := ERR_RESPONSE_ID;
                     statFBState :=  LAcycCom_ReadWriteStatus#FB_ERROR;

                     // Error : The received number of parameters does NOT match with the requested number of parameters
                   ELSIF  (statCmdBusy = FALSE) AND
                     (TO_INT(statRespParameter.header.parameterNo) <> 1) AND
                      (tempCmdValid = TRUE) THEN

                     statStateNumber := statFBSubState;
                     statStatus := ERR_PARAMETER_NO;
                     statFBState :=  LAcycCom_ReadWriteStatus#FB_ERROR;

                     // Error : The drive object does NOT match with the responsed DO
                   ELSIF  (statCmdBusy = FALSE) AND
                      (TO_BYTE(statDoId) <> statRespParameter.header.doId) AND
                      (tempCmdValid = TRUE) THEN

                     statStateNumber := statFBSubState;
                     statStatus := ERR_DRIVE_OBJECT_NO;
                     statFBState :=  LAcycCom_ReadWriteStatus#FB_ERROR;

                     // No error occurred during reading parameters
                   ELSIF  (tempCmdValid = TRUE) THEN
                     // Analyse of the response buffer
                     statParameter[0].format := statRespParameter.data[0];  // Format of the parameter

                     // Format = Error
                     IF (((TO_SINT (statRespParameter.data[0]) > FORMAT_DOUBLE_WORD) OR
                       ((TO_SINT (statRespParameter.data[0]) > FORMAT_FLOATING_POINT) AND (TO_SINT (statRespParameter.data[0]) < FORMAT_OCTET_STRING)) OR
                       ((TO_SINT (statRespParameter.data[0]) > FORMAT_OCTET_STRING) AND (TO_SINT (statRespParameter.data[0]) < FORMAT_TIME_DIFFERENCE)) OR
                       ((TO_SINT (statRespParameter.data[0]) > FORMAT_TIME_DIFFERENCE) AND (TO_SINT (statRespParameter.data[0]) < FORMAT_BYTE)) OR
                       (TO_SINT (statRespParameter.data[0]) < FORMAT_INTEGER_8))) AND (TO_SINT (statRespParameter.data[0]) <> FORMAT_ZERO)
                     THEN

                       // Format = Error, summarize the first and second error BYTE in a WORD error variable for each parameter
                       statParameter[0].errorValue := statRespParameter.data[3];
                       statParameter[0].dwordValue := DWORD#16#0;
                       statParameter[0].realValue := REAL#0.0;
                       statdiagnostics.errorValue := statParameter[0].errorValue; // V1.3.2

                       IF  (statFirstParameterError = NO_PARAMETER_ERROR) THEN
                         statdiagnostics.firstParameterError := 0;
                         statFirstParameterError := 0;

                         statStateNumber := statFBSubState;
                         statStatus := ERR_PARAMETER;
                         statFBState :=  LAcycCom_ReadWriteStatus#FB_ERROR;
                       END_IF;

                     ELSE
                       CASE TO_SINT (statRespParameter.data[0]) OF
                         FORMAT_INTEGER_8:
                           statParameter[0].realValue := TO_REAL(TO_SINT (statRespParameter.data[2]));
                           statParameter[0].dwordValue := statRespParameter.data[2];
                           statParameter[0].errorValue := BYTE#16#FF; // Sets the error status and diagnostics

                         FORMAT_INTEGER_16:
                           tempWord.%B0 := statRespParameter.data[3];
                           tempWord.%B1 := statRespParameter.data[2];

                           statParameter[0].realValue := TO_REAL(TO_INT (tempWord));
                           statParameter[0].dwordValue := tempWord;
                           statParameter[0].errorValue := BYTE#16#FF; // Sets the error status and diagnostics

                         FORMAT_INTEGER_32:
                           tempDWord.%B0 := statRespParameter.data[5];
                           tempDWord.%B1 := statRespParameter.data[4];
                           tempDWord.%B2 := statRespParameter.data[3];
                           tempDWord.%B3 := statRespParameter.data[2];

                           statParameter[0].realValue := TO_REAL(TO_DINT (tempDWord));
                           statParameter[0].dwordValue := tempDWord;
                           statParameter[0].errorValue := BYTE#16#FF; // Sets the error status and diagnostics

                         FORMAT_UNSIGNED_8, FORMAT_OCTET_STRING: // V1.5 change OCTET_STRING:
                           statParameter[0].realValue := TO_REAL(TO_USINT (statRespParameter.data[2]));
                           statParameter[0].dwordValue := statRespParameter.data[2];
                           statParameter[0].errorValue := BYTE#16#FF; // Sets the error status and diagnostics

                         FORMAT_UNSIGNED_16:
                           tempWord.%B0 := statRespParameter.data[3];
                           tempWord.%B1 := statRespParameter.data[2];

                           statParameter[0].realValue := TO_REAL(TO_UINT (tempWord));
                           statParameter[0].dwordValue := tempWord;
                           statParameter[0].errorValue := BYTE#16#FF; // Sets the error status and diagnostics

                         FORMAT_UNSIGNED_32, FORMAT_TIME_DIFFERENCE:
                           tempDWord.%B0 := statRespParameter.data[5];
                           tempDWord.%B1 := statRespParameter.data[4];
                           tempDWord.%B2 := statRespParameter.data[3];
                           tempDWord.%B3 := statRespParameter.data[2];

                           statParameter[0].realValue := TO_REAL(TO_UDINT (tempDWord));
                           statParameter[0].dwordValue := tempDWord;
                           statParameter[0].errorValue := BYTE#16#FF; // Sets the error status and diagnostics

                         FORMAT_FLOATING_POINT, FORMAT_DOUBLE_WORD:
                           tempDWord.%B0 := statRespParameter.data[5];
                           tempDWord.%B1 := statRespParameter.data[4];
                           tempDWord.%B2 := statRespParameter.data[3];
                           tempDWord.%B3 := statRespParameter.data[2];

                           statParameter[0].realValue := TO_REAL (tempDWord);
                           statParameter[0].dwordValue := tempDWord;
                           statParameter[0].errorValue := BYTE#16#FF; // Sets the error status and diagnostics

                         FORMAT_BYTE:
                           statParameter[0].realValue := TO_REAL(TO_DWORD (statRespParameter.data[2]));
                           statParameter[0].dwordValue := statRespParameter.data[2];
                           statParameter[0].errorValue := BYTE#16#FF; // Sets the error status and diagnostics

                         FORMAT_WORD:
                           tempWord.%B0 := statRespParameter.data[3];
                           tempWord.%B1 := statRespParameter.data[2];

                           statParameter[0].realValue := TO_REAL(TO_DWORD (tempWord));
                           statParameter[0].dwordValue := tempWord;
                           statParameter[0].errorValue := BYTE#16#FF; // Sets the error status and diagnostics

                         ELSE
                           ;
                       END_CASE;

                     END_IF; // Format = Error

                     statdiagnostics.errorValue := statParameter[0].errorValue;

                     statCmdBusy := FALSE;
                     statCmdError := FALSE;

                          // Next state is depending on the FB mode
                          IF NOT(statFBState = LAcycCom_ReadWriteStatus#FB_ERROR) THEN
                            statStatus := STATUS_RELEASE;
                            statFBState := LAcycCom_ReadWriteStatus#FB_RELEASE;

                          END_IF; // statMode = MODE_WITH_BUFFER_MANAGER
                   END_IF; // statCmdError = TRUE

                   LAcycCom_ReadWriteStatus#FB_BUSY_WAIT:
                   // Timer for temporary errors
                   instIECTimer(signal := statTimerStart,
                                 duration := TIMER_TEMP_ERROR);

                   statTimerStart := TRUE;
                   IF  (instIECTimer.output = TRUE) THEN
                     statTimerStart := FALSE;
                     statFBSubState := statFBSubStateOld;
                   END_IF;

                 ELSE

                   statStatus := ERR_UNDEFINED_SUBSTATE;
                   statStateNumber := statFBState;
                   statFBState :=  LAcycCom_ReadWriteStatus#FB_ERROR;
               END_CASE;

             ELSE

               statStatus := ERR_COMMAND_TIMEOUT;
               statStateNumber := statFBState;
               statFBState :=  LAcycCom_ReadWriteStatus#FB_ERROR;
             END_IF; // ( (buffer.element[statAllocatedIndex].enable = TRUE) AND  (statMode = MODE_WITH_BUFFER_MANAGER)) OR statMode = MODE_WITHOUT_BUFFER_MANAGER

        END_METHOD

        Method PUBLIC GetValueREAL : REAL
            GetValueREAL := statParameter[0].realValue;
        end_method

        Method PUBLIC GetValueDWORD : DWORD
            GetValueDWORD := statParameter[0].dwordValue;
        end_method

          //data type of driveobjectid has been changed from uint to int. This extra start method keeps compability to old versions of LAcycCom
          METHOD PUBLIC Start : BOOL
            VAR_INPUT
              driveObjectId : UINT;
              hardwareId    : HW_IO;
              parameterNumber: UINT;            // Number of the parameter
              index          : UINT;            // Parameter index
            END_VAR
            Start := THIS.Start(driveObjectId := TO_INT(driveObjectId), hardwareId := hardwareId, parameterNumber := parameterNumber, index := index);
          END_METHOD
          //data type of driveobjectid has been changed from uint to int. This extra start method can be used, if direct hw id is used and drive id object is not used (equivalent to driveobjectid = -1)
          METHOD PUBLIC Start : BOOL
            VAR_INPUT
              hardwareId    : HW_IO;
              parameterNumber: UINT;            // Number of the parameter
              index          : UINT;            // Parameter index
          END_VAR
          Start := THIS.Start(driveObjectId := -1, hardwareId := hardwareId, parameterNumber := parameterNumber, index := index);
        END_METHOD

        METHOD PUBLIC Start : BOOL
            VAR_INPUT
                driveObjectId  : INT := -1;   // Optional: Identification number of the drive object (value =0: driveObjectId is NOT used, i.e. the corresponding drive object is only addressed via the hardwareId)
                hardwareId : HW_IO;   // Hardware identifier of the hardware module
                parameterNumber : UINT;   // Number of the parameter
                index : UINT;   // Parameter index
             END_VAR

             statparameterNumber := parameterNumber;
             statindex := index;
             statDoId := driveObjectId;
             statHwId := hardwareId;

             // starts functionality
             IF NOT ((statFBState = LAcycCom_ReadWriteStatus#FB_IDLE OR
                 statFBState = LAcycCom_ReadWriteStatus#FB_DONE OR
                 statFBState = LAcycCom_ReadWriteStatus#FB_ERROR) AND
                 statrequestBuffer <> NULL) THEN
                   Start := FALSE;
             ELSE
               // Initialisation
               Start := TRUE;
               statAllocatedIndex := -1;
               statSubfunctionStatus :=  WORD#16#0000;
               statDataRecordNo := DINT#0;
               statStateNumber := LAcycCom_ReadWriteStatus#FB_IDLE;
               statDatasetType := SINT#0;
               statFirstParameterError := -1;
               statErrorCount := UINT#0;
               statFBSubState := LAcycCom_ReadWriteStatus#FB_BUSY_WRREC;
               statFBState := LAcycCom_ReadWriteStatus#FB_FIRST_CYCLE;

               instIECTimer(signal := FALSE,
                             duration := TIMER_ALLOCATION);

             END_IF;
        END_METHOD

    END_CLASS
END_NAMESPACE
